Fanuc KAREL source: kt00190.KL

-- PROVISIONAL review KL for V770-1; original PC SHA256 d2fd97ca40609077053aeab17203b83a83a60b6b4f6a193015d4684353332838
-- Incomplete behavior may be omitted. Consult companion uncertainty JSON. Do not deploy.
PROGRAM KT00190
%NOLOCKGROUP
VAR
  OUT : REAL
-- UNRESOLVED_DECL H1 type=002017
-- UNRESOLVED_DECL Y2 type=002018
BEGIN
  -- UNRESOLVED_PC offsets 5-19; opcodes 2E,22,9D,33,B4
  -- UNRESOLVED_PC offsets 24-38; opcodes 2E,22,9D,33,B2
  -- UNRESOLVED_PC offsets 43-69; opcodes 22,9D,33,B3,22,9D,33,B1,56,64,23
  -- UNRESOLVED_PC offsets 74-78; opcodes 7F
END KT00190
